{attribute 'GeneratedUsingTerminal: '}
{attribute addProperty BoxType ""}
{attribute addProperty Id "_defaultAT %I*SyncUnitTasks_5FDC977018"}
{attribute addProperty CRC "3282258768"}
{attribute addProperty Size "18"}
TYPE SyncUnits_C3A34B50 EXTENDS TcoIo.SyncUnitsBase_AD6C35CE :
STRUCT
	{attribute addProperty Name "_default"}
	_default : SyncUnitTasks_5FDC9770;
END_STRUCT
END_TYPE

(* stored: Version 1.2.0.0, ProductVersion 3.1.4024.11
   DUT SyncUnits_C3A34B50: Id {ae93b09f-9b05-080a-117d-4c72d787e2fe} *)
